// TIA Portal project "AWL LIBRO 9" (V11)

(* hardware
DEVICE "S7300/ET200 station_1"  SIMATIC 300-Station
   slot 0: "Perfil soporte_0"  Rail  6ES7 390-1***0-0AA0
   slot 2: "PLC_1"  CPU 313C-2 DP  6ES7 313-6CF03-0AB0  V2.6
      slot 0: "Interfaz MPI_1"  MPI
      slot 1: "Interfaz DP_1"  DP
      slot 2: "DI16/DO16_1"  DI16/DO16
      slot 4: "Contaje_1"  Counter
*)

// ===== PLC "PLC_1"  CPU 313C-2 DP =====

VAR_GLOBAL   // PLC tag table "Tabla de variables estándar"
   "PRESELECCION" AT %E0.0 : Bool;
   "EJECUCION" AT %E0.1 : Bool;
   "EMERGENCIA" AT %E0.2 : Bool;
   "S0" AT %E0.3 : Bool;
   "S1" AT %E0.4 : Bool;
   "S2" AT %E0.5 : Bool;
   "S3" AT %E0.6 : Bool;
   "S4" AT %E0.7 : Bool;
   "S5" AT %E1.0 : Bool;
   "MEZCLA 1" AT %A0.0 : Bool;
   "MEZCLA 2" AT %A0.1 : Bool;
   "MEZCLA 3" AT %A0.2 : Bool;
   "MEZCLA 4" AT %A0.3 : Bool;
   "MEZCLA 5" AT %A0.4 : Bool;
   "MEZCLA 6" AT %A0.5 : Bool;
   "CONTADOR" AT %MW10 : Int;
   "VALVULA A" AT %A1.0 : Bool;
   "VALVULA B" AT %A1.1 : Bool;
   "VALVULA C" AT %A1.2 : Bool;
   "HOMOGENIZADOR" AT %A1.3 : Bool;
   "SALIDAS PROCESO" AT %AB1 : Byte;
   "SALIDAS SELECCION" AT %AB0 : Byte;
   "T0" AT %T0 : Timer;
END_VAR

DATA_BLOCK "FLANCOS"   // DB1
{ S7_Optimized_Access := 'FALSE' }
VERSION : 0.1
   VAR
      F0 : Bool;
      F1 : Bool;
      F2 : Bool;
      F3 : Bool;
      F4 : Bool;
      F5 : Bool;
      F6 : Bool;
      F7 : Bool;
      F8 : Bool;
      F9 : Bool;
      F10 : Bool;
      F11 : Bool;
   END_VAR
BEGIN
END_DATA_BLOCK

ORGANIZATION_BLOCK "Main"   // OB1, STL
TITLE = EJERCICIO 9. / "Main Program Sweep (Cycle)"
{ S7_Optimized_Access := 'FALSE' }
VERSION : 0.1
   VAR_TEMP
      OB1_EV_CLASS : Byte;   // Bits 0-3 = 1 (Coming event), Bits 4-7 = 1 (Event class 1)
      OB1_SCAN_1 : Byte;   // 1 (Cold restart scan 1 of OB 1), 3 (Scan 2-n of OB 1)
      OB1_PRIORITY : Byte;   // Priority of OB Execution
      OB1_OB_NUMBR : Byte;   // 1 (Organization block 1, OB1)
      OB1_RESERVED_1 : Byte;   // Reserved for system
      OB1_RESERVED_2 : Byte;   // Reserved for system
      OB1_PREV_CYCLE : Int;   // Cycle time of previous OB1 scan (milliseconds)
      OB1_MIN_CYCLE : Int;   // Minimum cycle time of OB1 (milliseconds)
      OB1_MAX_CYCLE : Int;   // Maximum cycle time of OB1 (milliseconds)
      OB1_DATE_TIME : Date_And_Time;   // Date and time OB1 started
   END_VAR
BEGIN
END_ORGANIZATION_BLOCK